// TIA Portal V18 export
// export: Created 2026-06-08T16:04:36.7781472Z, ExportSetting WithDefaults, DisplayName Totally Integrated Automation Portal, DisplayVersion V18, DisplayName TIA Portal Openness, DisplayVersion V18, DisplayName TIA Portal Version Control Interface, DisplayVersion V18, DisplayName STEP 7 Professional, DisplayVersion V18, DisplayName STEP 7 Safety, DisplayVersion V18, DisplayName WinCC Professional, DisplayVersion V18
VAR_GLOBAL   // PLC tag table "INPUT_M"
   M_Mode AT %M10.0 : Bool;   // Switch chế độ 1 auto, 0 manu
   M_CB_Cao AT %M10.1 : Bool;   // Cảm biến sản phẩm cao
   M_CB_Trung_Binh AT %M10.2 : Bool;   // Cảm biến sản phẩm trung bình
   M_CB_Thap AT %M10.3 : Bool;   // Cảm biến sản phẩm thấp
   M_BT AT %M10.4 : Bool;   // Chạy/Dừng động cơ băng tải
   M_Xylanh_Cao AT %M10.5 : Bool;   // Đóng/mở xi lanh sản phẩm cao
   M_Xylanh_TB AT %M10.6 : Bool;   // Đóng/mở xi lanh sản phẩm trung bình
END_VAR
